KUKA KRL program: BrakeTest.src, BrakeTest.dat

--- BrakeTest.src ---
&ACCESS RVP
&REL 1
&COMMENT BRAKE TEST
&PARAM EDITMASK = *
DEF BrakeTest( )
;FOLD INI
  ;FOLD BASISTECH INI
    GLOBAL INTERRUPT DECL 3 WHEN $STOPMESS==TRUE DO IR_STOPM ( )
    INTERRUPT ON 3
    BAS (#INITMOV,0 )
  ;ENDFOLD (BASISTECH INI)
  ;FOLD USER INI
    ;Make your modifications here

  ;ENDFOLD (USER INI)
;ENDFOLD (INI)

  ;******************************;
  ;         TESLA MOTORS         ;
  ;ALL MODELS                    ;
  ;Program 08                    ;
  ;Brake Test Program            ;
  ;Template    KRC4.V7.1         ;
  ;******************************;

;Brake Test Request Program

braketestreq ( )



END

--- BrakeTest.dat ---
&ACCESS RVP
&REL 1
&COMMENT BRAKE TEST
&PARAM EDITMASK = *
DEFDAT BrakeTest
;FOLD EXTERNAL DECLARATIONS;%{PE}%MKUKATPBASIS,%CEXT,%VCOMMON,%P
;FOLD BASISTECH EXT;%{PE}%MKUKATPBASIS,%CEXT,%VEXT,%P
EXT  BAS (BAS_COMMAND  :IN,REAL  :IN )
DECL INT SUCCESS
;ENDFOLD (BASISTECH EXT)
;FOLD USER EXT;%{E}%MKUKATPUSER,%CEXT,%VEXT,%P
;Make here your modifications

;ENDFOLD (USER EXT)
;ENDFOLD (EXTERNAL DECLARATIONS)
ENDDAT
